TYPE stUnderPressureTestStatus_V2 :
STRUCT
	bError		: BOOL;
	bBusy		: BOOL;
	bWorkEnd 	: BOOL;
	bWorkAllow	: BOOL;
	bManual		: BOOL;
	bResetSequence	: BOOL;
END_STRUCT
END_TYPE

(* stored: Version 1.1.0.1, ProductVersion 3.1.4024.13
   DUT stUnderPressureTestStatus_V2: Id {d5cf9997-5488-45e0-bc06-f98f08996b49} *)
